// TIA Portal V20 export
TYPE "PartStatus1"
// stored: Access Published
   STRUCT
      noPart : Bool;
      okPart : Bool;
      nokPart : Bool;
      gaugePart : Bool;
      InsepctionPart : Bool;
      sampledPart : Bool;
      Reserved_0 : Bool;
      Reserved_1 : Bool;
   END_STRUCT;
END_TYPE
